Omron Sysmac Studio project 20-801-IP106 (Sysmac Studio 1.41.0.10, StandardProject)

# Controller new_Controller_0: NX1P2-1040DT version 1.41
Units and slaves: 節點1 : ASDA-A2-E CoE Drive (E001); 節點2 : ASDA-A2-E CoE Drive (E002); 節點3 : ASDA-A2-E CoE Drive (E003); 節點4 : ASDA-A2-E CoE Drive (E004)
Axis MC_AxisX, settings changed from default: AxisType=ServoType, FunctionLimit=SingleAxisPTP, UnitsConversion=EnumElement2, UnitsNumerator=1280000, UnitsDenominator=20, MaxVelocity=1500, MaxJogVelocity=150, InPositionBand=1, InPositionCheckTime=100, ZeroPositionBand=0.01, HomingMode=LimitOnly, StartDirection=NegativeDirection, HomingVelocity=10, HomingApproachVelocity=5, OriginCompensationValue=1, CompensationVelocity=5
Axis MC_AxisY, settings changed from default: AxisNumber=1, AxisType=ServoType, FunctionLimit=SingleAxisPTP, UnitsConversion=EnumElement2, UnitsNumerator=1280000, UnitsDenominator=20, MaxVelocity=1500, MaxJogVelocity=150, InPositionBand=1, InPositionCheckTime=100, ZeroPositionBand=0.01, HomingMode=LimitOnly, StartDirection=NegativeDirection, HomingVelocity=10, HomingApproachVelocity=5, OriginCompensationValue=1, CompensationVelocity=5
Axis MC_AxisZ, settings changed from default: AxisNumber=2, AxisType=ServoType, FunctionLimit=SingleAxisPTP, UnitsConversion=EnumElement2, UnitsNumerator=1280000, UnitsDenominator=20, MaxVelocity=1500, MaxJogVelocity=150, InPositionBand=1, InPositionCheckTime=100, ZeroPositionBand=0.01, HomingMode=LimitOnly, StartDirection=NegativeDirection, HomingVelocity=10, HomingApproachVelocity=5, OriginCompensationValue=1, CompensationVelocity=5
Axis MC_AxisS, settings changed from default: AxisNumber=3, AxisType=ServoType, UnitsConversion=EnumElement5, UnitsNumerator=1280000, UnitsDenominator=120, TravelDistancePerWorkRotation=360, WorkGearRatio=3, MaxVelocity=18000, MaxJogVelocity=1800, InPositionBand=0.1, InPositionCheckTime=500, ZeroPositionBand=0.05, HomingVelocity=100, HomingApproachVelocity=50
Task PrimaryTask (priority 4, period or condition 2000): prAxisDefineX, prAxisDefineY, prAxisDefineZ, prAxisDefineS, prCommProgram, prError, prInitialize, prScrewData, prBZAndLight, prBowlFeeder, prCycleTime, prMain, prScrewFlow, prFeedScrew

TYPE stScrewData : STRUCT
    PositionX : array[0..29] of lreal;
    PositionY : array[0..29] of lreal;
    PositionZ : array[0..29] of lreal;
    IsLastPoint : array[0..29] of bool;
END_STRUCT END_TYPE
TYPE AxisShow : STRUCT
    bHomed : BOOL;
END_STRUCT END_TYPE

VAR_GLOBAL CONSTANT
    MC_AxisX : _sAXIS_REF;  (* at MC://_MC_AX[0] *)
    MC_AxisY : _sAXIS_REF;  (* at MC://_MC_AX[1] *)
    MC_AxisZ : _sAXIS_REF;  (* at MC://_MC_AX[2] *)
    MC_AxisS : _sAXIS_REF;  (* at MC://_MC_AX[3] *)
END_VAR
VAR_GLOBAL
    PB_Start : BOOL;  (* at BuiltInIO://cpu/#0/Input_Bit_00; published *)
    PB_Reset : BOOL;  (* at BuiltInIO://cpu/#0/Input_Bit_01; published *)
    PB_ESTOP : BOOL;  (* at BuiltInIO://cpu/#0/Input_Bit_02; published *)
    LS_UpDownBack : BOOL;  (* at BuiltInIO://cpu/#0/Input_Bit_03; published *)
    LS_UpDownOut : BOOL;  (* at BuiltInIO://cpu/#0/Input_Bit_04; published *)
    LS_THBack : BOOL;  (* at BuiltInIO://cpu/#0/Input_Bit_05; published *)
    LS_THOut : BOOL;  (* at BuiltInIO://cpu/#0/Input_Bit_06; published *)
    SNR_AirSource : BOOL;  (* at BuiltInIO://cpu/#0/Input_Bit_07; published *)
    SNR_FeedScrew : BOOL;  (* at BuiltInIO://cpu/#0/Input_Bit_08; published *)
    SNR_BowlFeeder : BOOL;  (* at BuiltInIO://cpu/#0/Input_Bit_09; published *)
    SNR_InPositionCheck : BOOL;  (* at BuiltInIO://cpu/#0/Input_Bit_10; published *)
    SOL_UpDown : BOOL;  (* at BuiltInIO://cpu/#0/Output_Bit_00; published *)
    SOL_TH : BOOL;  (* at BuiltInIO://cpu/#0/Output_Bit_01; published *)
    SOL_Fix : BOOL;  (* at BuiltInIO://cpu/#0/Output_Bit_02; published *)
    SOL_FeedScrew : BOOL;  (* at BuiltInIO://cpu/#0/Output_Bit_03; published *)
    BZ : BOOL;  (* at BuiltInIO://cpu/#0/Output_Bit_04; published *)
    YL : BOOL;  (* at BuiltInIO://cpu/#0/Output_Bit_10; published *)
    GL : BOOL;  (* at BuiltInIO://cpu/#0/Output_Bit_06; published *)
    RL : BOOL;  (* at BuiltInIO://cpu/#0/Output_Bit_07; published *)
    RY_BowlFeeder : BOOL;  (* at BuiltInIO://cpu/#0/Output_Bit_08; published *)
    RY_BrakeAxisZ : BOOL;  (* at BuiltInIO://cpu/#0/Output_Bit_09; published *)
    RY_BowlFeederMotor : BOOL;  (* at IOBus://unit#3/Output Bit 16 bits/Output Bit 00; published *)
    AutoStatus : BOOL;  (* published *)
    HMIPB_AllSerchHome : BOOL;  (* published *)
    HMIPB_UpDown : BOOL;  (* published *)
    HMIPB_TH : BOOL;  (* published *)
    HMIPB_Fix : BOOL;  (* published *)
    HMIPB_ScrewMode_Torque : BOOL;  (* 鎖付方式(扭力/位置); published *)
    HMIPB_FeedScrew : BOOL;  (* published *)
    HMIPB_HighSpeed : BOOL;  (* published *)
    HMIPB_AlarmResetAxisX : BOOL;  (* published *)
    HMIPB_AlarmResetAxisY : BOOL;  (* published *)
    HMIPB_AlarmResetAxisZ : BOOL;  (* published *)
    HMIPB_AlarmResetAxisS : BOOL;  (* published *)
    HMIPB_ServoStopAxisX : BOOL;  (* published *)
    HMIPB_ServoStopAxisY : BOOL;  (* published *)
    HMIPB_ServoStopAxisZ : BOOL;  (* published *)
    HMIPB_ServoStopAxisS : BOOL;  (* published *)
    HMIPB_FW_AxisX : BOOL;  (* published *)
    HMIPB_RW_AxisX : BOOL;  (* published *)
    HMIPB_FW_AxisY : BOOL;  (* published *)
    HMIPB_RW_AxisY : BOOL;  (* published *)
    HMIPB_FW_AxisZ : BOOL;  (* published *)
    HMIPB_RW_AxisZ : BOOL;  (* published *)
    HMIPB_FW_AxisS : BOOL;  (* published *)
    HMIPB_RW_AxisS : BOOL;  (* published *)
    HMIPB_ServoON_AxisX : BOOL;  (* published *)
    HMIPB_ServoON_AxisY : BOOL;  (* published *)
    HMIPB_ServoON_AxisZ : BOOL;  (* published *)
    HMIPB_ServoON_AxisS : BOOL;  (* published *)
    HMIPB_SerchHome_AxisX : BOOL;  (* published *)
    HMIPB_SerchHome_AxisY : BOOL;  (* published *)
    HMIPB_SerchHome_AxisZ : BOOL;  (* published *)
    HMIPB_SerchHome_AxisS : BOOL;  (* published *)
    HMIPB_MoveAbs_AxisX : BOOL;  (* published *)
    HMIPB_MoveAbs_AxisY : BOOL;  (* published *)
    HMIPB_MoveAbs_AxisZ : BOOL;  (* published *)
    HMIPB_GoZero_AxisX : BOOL;  (* published *)
    HMIPB_GoZero_AxisY : BOOL;  (* published *)
    HMIPB_GoZero_AxisZ : BOOL;  (* published *)
    HMIPB_MoveAbs_TechX : BOOL;  (* published *)
    HMIPB_MoveAbs_TechY : BOOL;  (* published *)
    HMIPB_MoveAbs_TechZ : BOOL;  (* published *)
    HMIPB_ResetCount : BOOL;  (* published *)
    HMIPB_BrakeAxisZ : BOOL;  (* published *)
    ReadScrewData : BOOL;  (* published *)
    WriteScrewData : BOOL;  (* published *)
    SetPointData : BOOL;  (* published *)
    Error_PB_ESTOP : BOOL;  (* published *)
    Error_LS_UpDownBack : BOOL;  (* published *)
    Error_LS_UpDownOut : BOOL;  (* published *)
    Error_LS_THBack : BOOL;  (* published *)
    Error_LS_THOut : BOOL;  (* published *)
    Error_SNR_AirSource : BOOL;  (* published *)
    Error_SNR_FeedScrew : BOOL;  (* published *)
    Error_SNR_BowlFeeder : BOOL;  (* published *)
    Error_AxisX : BOOL;  (* published *)
    Error_AxisY : BOOL;  (* published *)
    Error_AxisZ : BOOL;  (* published *)
    Error_AxisS : BOOL;  (* published *)
    Flash1s : BOOL;
    SystemReadyStatus : BOOL;
    ErrorStatus_MachineStop : BOOL;  (* published *)
    ErrorStatus_MachineNonStop : BOOL;  (* published *)
    MachineRunning : BOOL;  (* published *)
    UP_InitialFlag : BOOL;
    FixOff_InitialFlag : BOOL;
    ScrewStopFlag : BOOL;
    SerchHomeAxisX_InitialFlag : BOOL;
    SerchHomeAxisY_InitialFlag : BOOL;
    SerchHomeAxisZ_InitialFlag : BOOL;
    SerchHomeAxisS_InitialFlag : BOOL;
    GoZeroAxisX_InitialFlag : BOOL;
    GoZeroAxisY_InitialFlag : BOOL;
    GoZeroAxisZ_InitialFlag : BOOL;
    Main2ScrewFlag : BOOL;  (* Main發screw開始flag *)
    Main2FeedScrewFlag : BOOL;  (* Main發送螺絲開始flag *)
    Main2DownFlag : BOOL;
    Main2UpFlag : BOOL;
    FeedScrewErrorFlag : BOOL;
    ResetFeedScrewErrorFlag : BOOL;
    ScrewNGFlag : BOOL;
END_VAR
VAR_GLOBAL RETAIN
    ScrewDatas : array[0..39] of stscrewdata;
    HMI_ItemNotExistsDelayTime : LINT;  (* published *)
    HMI_ItemExistsDelayTime : LINT;  (* published *)
    HMI_ItemNotExistsErrorTime : LINT;  (* published *)
    HMI_FeedScrewTime : LINT;  (* published *)
    HMI_CheckOKTime : LINT;  (* 滑牙計時OK; published *)
    HMI_CheckNGTime : LINT;  (* 滑牙計時NG; published *)
    HMI_AutoSpeedXY : LREAL;  (* mm/s; published *)
    HMI_AutoSpeedZ : LREAL;  (* mm/s; published *)
    HMI_HighSpeed : LREAL;  (* mm/s; published *)
    HMI_LowSpeed : LREAL;  (* mm/s; published *)
    HMI_ScrewSpeed : LREAL;  (* RPM; published *)
    HMI_ScrewTorque : LREAL;  (* %; published *)
END_VAR
VAR_GLOBAL
    HMI_Acc : LREAL;
    HMI_Dec : LREAL;
    HMI_Jerk : LREAL;
END_VAR
VAR_GLOBAL RETAIN
    HMI_JobNo : INT;  (* published *)
    HMI_PointNo : INT;  (* published *)
    HMI_AllCount : UDINT;  (* published *)
END_VAR
VAR_GLOBAL
    HMI_CycleTime : LINT;  (* published *)
END_VAR
VAR_GLOBAL RETAIN
    HMI_BackoutD : LREAL;  (* published *)
    ScrewInClip : INT;
    OilPointX : LREAL;  (* published *)
    OilPointY : LREAL;  (* published *)
    OilPointZ : LREAL;  (* published *)
END_VAR
VAR_GLOBAL
    PositionX : ARRAY[0..29] of lreal;  (* published *)
    PositionY : ARRAY[0..29] of lreal;  (* published *)
    PositionZ : ARRAY[0..29] of lreal;  (* published *)
    LastScrewPoint : ARRAY[0..29] of bool;  (* published *)
    ShowOKs : ARRAY[0..29] of bool;  (* published *)
    ShowNGs : ARRAY[0..29] of bool;  (* published *)
    Homed_ShowAixs : array[0..3] of bool;  (* published *)
    Error_ShowAixs : array[0..3] of bool;  (* published *)
    POT_ShowAxis : array[0..3] of bool;  (* published *)
    NOT_ShowAxis : array[0..3] of bool;  (* published *)
    CurrentPostion_ShowAxis : array[0..3] of lreal;  (* published *)
    CurrentSpeed_ShowAxis : array[0..3] of lreal;  (* published *)
    CurrentTorque_ShowAxis : array[0..3] of lreal;  (* published *)
    SOL_BowlFeederBlow : BOOL;  (* at IOBus://unit#3/Output Bit 16 bits/Output Bit 01 *)
END_VAR

PROGRAM prCommProgram
VAR
    statusFlash1s : BOOL;
    bClock : BOOL;
    TON1 : TON;
    TON2 : TON;
    R_TRIG1 : R_TRIG;
END_VAR
VAR_EXTERNAL
    Flash1s : BOOL;
    HMIPB_ResetCount : BOOL;
    HMI_AllCount : UDINT;
END_VAR
//bClock:=Get1sClk();
IF HMIPB_ResetCount THEN
	HMI_AllCount:=0;
END_IF;
//flsash 1s
TON1(In:=NOT(statusFlash1s), PT:=t#1s);
TON2(In:=(statusFlash1s), PT:=t#1s);
IF TON1.Q THEN
	bClock:=TRUE;
END_IF;
IF TON2.Q THEN
	bClock:=FALSE;
END_IF;
Flash1s:=bClock;
statusFlash1s:=Flash1s;
END_PROGRAM

PROGRAM prBowlFeeder
VAR
    bowlfedder1 : BowlFeeder;
END_VAR
VAR_EXTERNAL
    SNR_BowlFeeder : BOOL;
    HMI_ItemNotExistsDelayTime : LINT;
    HMI_ItemExistsDelayTime : LINT;
    HMI_ItemNotExistsErrorTime : LINT;
    RY_BowlFeeder : BOOL;
    Error_SNR_BowlFeeder : BOOL;
    SOL_BowlFeederBlow : BOOL;
    RY_BowlFeederMotor : BOOL;
END_VAR
bowlfedder1(
	bFullSNR:=SNR_BowlFeeder,
	iItemNotExistDelayTime:=HMI_ItemNotExistsDelayTime,
	iItemExistTime:=HMI_ItemExistsDelayTime,
	iItemNotExistErrorTime:=HMI_ItemNotExistsErrorTime,
	bFullSNRError=>Error_SNR_BowlFeeder);
RY_BowlFeeder:=bowlfedder1.bFullRY;
RY_BowlFeederMotor:=bowlfedder1.bFullRY;
SOL_BowlFeederBlow:=bowlfedder1.bFullRY;
END_PROGRAM

PROGRAM prInitialize
VAR
    InitFlow : INT;
    TON1 : TON;
    R_TRIG1 : R_TRIG;
    ErrorState : BOOL;
END_VAR
VAR_EXTERNAL
    ErrorStatus_MachineStop : BOOL;
    PB_Reset : BOOL;
    LS_UpDownBack : BOOL;
END_VAR
VAR_EXTERNAL CONSTANT
    MC_AxisZ : _sAXIS_REF;
    MC_AxisS : _sAXIS_REF;
    MC_AxisX : _sAXIS_REF;
    MC_AxisY : _sAXIS_REF;
END_VAR
VAR_EXTERNAL
    HMIPB_ServoON_AxisX : BOOL;
    HMIPB_ServoON_AxisY : BOOL;
    HMIPB_ServoON_AxisZ : BOOL;
    HMIPB_ServoON_AxisS : BOOL;
    SystemReadyStatus : BOOL;
    UP_InitialFlag : BOOL;
    SerchHomeAxisZ_InitialFlag : BOOL;
    GoZeroAxisZ_InitialFlag : BOOL;
    SerchHomeAxisX_InitialFlag : BOOL;
    SerchHomeAxisY_InitialFlag : BOOL;
    GoZeroAxisX_InitialFlag : BOOL;
    GoZeroAxisY_InitialFlag : BOOL;
    SerchHomeAxisS_InitialFlag : BOOL;
    FixOff_InitialFlag : BOOL;
    LS_THBack : BOOL;
    SOL_Fix : BOOL;
    HMIPB_AllSerchHome : BOOL;
    RY_BrakeAxisZ : BOOL;
    AutoStatus : BOOL;
    Error_AxisX : BOOL;
    Error_AxisY : BOOL;
    Error_AxisZ : BOOL;
    Error_AxisS : BOOL;
    Error_LS_THBack : BOOL;
    Error_LS_THOut : BOOL;
    Error_LS_UpDownBack : BOOL;
    Error_LS_UpDownOut : BOOL;
    Error_PB_ESTOP : BOOL;
    HMIPB_HighSpeed : BOOL;
    SOL_UpDown : BOOL;
    HMI_PointNo : INT;
END_VAR
//********************************************************************
//power on=0
//idle=1
//Servo On=2
//sol up=3
//up  reached=4

//Z軸未HOMED=100
//Axis Z serch home start=101
//Axis z serch home finiish=102

//Z軸已HOMED=200
//Axis Z go to 0 start=201
//Axis Z go to 0 finish=202

//X or Y軸未HOMED=300
//Axis X,Y serch home start=301
//Axis X,Y serch home finish=302

//X and Y軸已HOMED=400
//Axis X,Y go to 0 start=401
//Axis X,Y go to 0 finish=402

//Axis S serch home start=5
//Axis S serch home finish=6
//sol Fix off=7
//sol fix reached,system ready on=8
//********************************************************************
ErrorState:=
Error_AxisX OR
Error_AxisY OR
Error_AxisZ OR
Error_AxisS OR
Error_LS_THBack OR
Error_LS_THOut;
//power on=0
IF P_First_Run OR ErrorState OR R_TRIG1.Q THEN
	InitFlow:=0;
	SystemReadyStatus:=FALSE;
	AutoStatus:=FALSE;
	UP_InitialFlag:=FALSE;
	FixOff_InitialFlag:=FALSE;
	HMI_PointNo:=0;
END_IF;
//idle=1
IF InitFlow=0 AND NOT(ErrorState) THEN
	InitFlow:=1;
END_IF;
IF Error_PB_ESTOP THEN
	InitFlow:=1;
	AutoStatus:=FALSE;
	UP_InitialFlag:=FALSE;
	FixOff_InitialFlag:=FALSE;
END_IF;
//Servo On=2
R_TRIG1(Clk:=HMIPB_AllSerchHome);
TON1(In:=InitFlow=1 AND MC_AxisX.DrvStatus.MainPower AND MC_AxisY.DrvStatus.MainPower AND MC_AxisZ.DrvStatus.MainPower AND MC_AxisS.DrvStatus.MainPower, PT:=t#3s);
IF InitFlow=1 AND TON1.Q  and NOT(ErrorState) AND NOT(Error_PB_ESTOP) THEN
	HMIPB_ServoON_AxisX:=TRUE;
	HMIPB_ServoON_AxisY:=TRUE;
	HMIPB_ServoON_AxisZ:=TRUE;
	HMIPB_ServoON_AxisS:=TRUE;
	HMIPB_HighSpeed:=TRUE;
	InitFlow:=2;
END_IF;
//sol up=3
IF InitFlow=2 AND HMIPB_HighSpeed AND MC_AxisX.Status.Ready AND MC_AxisY.Status.Ready AND MC_AxisZ.Status.Ready AND MC_AxisS.Status.Ready AND RY_BrakeAxisZ THEN
	InitFlow:=3;
	UP_InitialFlag:=TRUE;
END_IF;
//up  reached=4
IF InitFlow=3 AND UP_InitialFlag AND LS_UpDownBack AND NOT(SOL_UpDown) THEN
	InitFlow:=4;
	UP_InitialFlag:=FALSE;
END_IF;
//********************************************************************
//Z軸未HOMED=100
IF InitFlow=4 AND NOT(UP_InitialFlag) AND NOT(MC_AxisZ.Details.Homed) THEN
	InitFlow:=100;
END_IF;
//Axis Z serch home start=101
IF InitFlow=100 THEN
	InitFlow:=101;
	SerchHomeAxisZ_InitialFlag:=TRUE;
END_IF;
//Axis z serch home finiish=102
IF InitFlow=101 AND NOT(SerchHomeAxisZ_InitialFlag) AND MC_AxisZ.Details.Homed THEN
	InitFlow:=102;
END_IF;
//********************************************************************
//Z軸已HOMED=200
IF InitFlow=4 AND NOT(UP_InitialFlag) AND MC_AxisZ.Details.Homed THEN
	InitFlow:=200;
END_IF;
//Axis Z go to 0 start=201
IF InitFlow=200 THEN
	InitFlow:=201;
	GoZeroAxisZ_InitialFlag:=TRUE;
END_IF;
//Axis Z go to 0 finish=202
IF InitFlow=201 AND NOT(GoZeroAxisZ_InitialFlag) AND MC_AxisZ.Details.InHome THEN
	InitFlow:=202;
END_IF;
//********************************************************************
//X or Y軸未HOMED=300
IF (InitFlow=102 OR InitFlow=202) AND (NOT(MC_AxisX.Details.Homed) OR NOT(MC_AxisY.Details.Homed)) THEN
	InitFlow:=300;
END_IF;
//Axis X,Y serch home start=301
IF InitFlow=300 THEN
	InitFlow:=301;
	SerchHomeAxisX_InitialFlag:=TRUE;
	SerchHomeAxisY_InitialFlag:=TRUE;
END_IF;
//Axis X,Y serch home finish=302
IF InitFlow=301 AND NOT(SerchHomeAxisX_InitialFlag) AND NOT(SerchHomeAxisY_InitialFlag) AND MC_AxisX.Details.Homed AND MC_AxisY.Details.Homed THEN
	InitFlow:=302;
END_IF;
//********************************************************************
//X and Y軸已HOMED=400
IF (InitFlow=102 OR InitFlow=202) AND MC_AxisX.Details.Homed AND MC_AxisY.Details.Homed THEN
	InitFlow:=400;
END_IF;
//Axis X,Y go to 0 start=401
IF InitFlow=400 THEN
	InitFlow:=401;
	GoZeroAxisX_InitialFlag:=TRUE;
	GoZeroAxisY_InitialFlag:=TRUE;
END_IF;
//Axis X,Y go to 0 finish=402
IF InitFlow=401 AND NOT(GoZeroAxisX_InitialFlag) AND NOT(GoZeroAxisY_InitialFlag) AND
	MC_AxisX.Details.InHome AND
	MC_AxisY.Details.InHome THEN
	InitFlow:=402;
END_IF;
//********************************************************************
//Axis S serch home start=5
IF InitFlow=302 AND MC_AxisX.Details.Homed  AND MC_AxisY.Details.Homed THEN
	InitFlow:=5;
	SerchHomeAxisS_InitialFlag:=TRUE;
END_IF;
IF InitFlow=402 AND MC_AxisX.Details.InHome AND MC_AxisY.Details.InHome THEN
	InitFlow:=5;
	SerchHomeAxisS_InitialFlag:=TRUE;
END_IF;
//Axis S serch home finish=6
IF InitFlow=5 AND NOT(SerchHomeAxisS_InitialFlag) AND MC_AxisS.Details.Homed THEN
	InitFlow:=6;
END_IF;
//sol Fix off=7
IF InitFlow=6 THEN
	InitFlow:=7;
	FixOff_InitialFlag:=TRUE;
END_IF;
//sol fix reached,system ready on=8
IF InitFlow=7 AND FixOff_InitialFlag AND NOT(SOL_Fix) THEN
	InitFlow:=8;
	FixOff_InitialFlag:=FALSE;
	SystemReadyStatus:=TRUE;
END_IF;
//Serch home finish=1000
IF InitFlow=8 AND SystemReadyStatus THEN
	InitFlow:=1000;
END_IF;
END_PROGRAM

PROGRAM prAxisDefineX
VAR
    MC_Power1 : MC_Power;
    MC_Reset1 : MC_Reset;
    MC_Stop1 : MC_Stop;
    MC_Home1 : MC_Home;
    MC_MoveJog1 : MC_MoveJog;
    MC_MoveAbsolute1 : MC_MoveAbsolute;
    MC_MoveAbsolute2 : MC_MoveAbsolute;
    MC_MoveAbsolute3 : MC_MoveAbsolute;
    MoveSpeed : LREAL;
    bInterlock : BOOL;
END_VAR
VAR_EXTERNAL CONSTANT
    MC_AxisX : _sAXIS_REF;
END_VAR
VAR_EXTERNAL
    HMIPB_ServoON_AxisX : BOOL;
    Error_AxisX : BOOL;
    HMIPB_SerchHome_AxisX : BOOL;
    SerchHomeAxisx_InitialFlag : BOOL;
    PB_Reset : BOOL;
    HMIPB_AlarmResetAxisX : BOOL;
    AutoStatus : BOOL;
    HMIPB_HighSpeed : BOOL;
    HMI_HighSpeed : LREAL;
    HMI_LowSpeed : LREAL;
    HMIPB_MoveAbs_AxisX : BOOL;
    GoZeroAxisX_InitialFlag : BOOL;
    HMIPB_FW_AxisX : BOOL;
    HMIPB_RW_AxisX : BOOL;
    PB_ESTOP : BOOL;
    HMIPB_ServoStopAxisX : BOOL;
    Homed_ShowAixs : array[0..3] of bool;
    Error_ShowAixs : array[0..3] of bool;
    POT_ShowAxis : array[0..3] of bool;
    NOT_ShowAxis : array[0..3] of bool;
    CurrentPostion_ShowAxis : array[0..3] of lreal;
    CurrentSpeed_ShowAxis : array[0..3] of lreal;
    CurrentTorque_ShowAxis : array[0..3] of lreal;
END_VAR
VAR_EXTERNAL CONSTANT
    MC_AxisZ : _sAXIS_REF;
END_VAR
VAR_EXTERNAL
    HMI_AutoSpeedXY : LREAL;
    HMIPB_GoZero_AxisX : BOOL;
    ScrewDatas : array[0..39] of stscrewdata;
    HMI_JobNo : INT;
    HMI_PointNo : INT;
    LS_UpDownBack : BOOL;
    SOL_UpDown : BOOL;
END_VAR
VAR_EXTERNAL CONSTANT
    _MC_ErrSta : WORD;
END_VAR
VAR_EXTERNAL
    HMI_Acc : LREAL;
    HMI_Dec : LREAL;
    HMI_Jerk : LREAL;
    HMIPB_MoveAbs_TechX : BOOL;
    PositionX : ARRAY[0..29] of lreal;
END_VAR
Error_AxisX:=MC_AxisX.DrvStatus.DrvAlarm OR MC_AxisX.DrvStatus.DrvWarning OR NOT(MC_AxisX.DrvStatus.MainPower) OR _MC_ErrSta<>0;		//Error
bInterlock:=MC_AxisX.DrvStatus.ServoOn AND MC_AxisZ.Details.Homed AND MC_AxisZ.Act.Pos>-1 AND MC_AxisZ.Act.Pos<1 AND LS_UpDownBack AND NOT(SOL_UpDown);
MC_Power1(Axis:=MC_AxisX, Enable:=HMIPB_ServoON_AxisX);		//servo on
MC_Reset1(Axis:=MC_AxisX, Execute:=HMIPB_AlarmResetAxisX OR PB_Reset);		//Alarm Reset
MC_Stop1(Axis:=MC_AxisX, Execute:=NOT(PB_ESTOP) OR HMIPB_ServoStopAxisX, Deceleration:=0, Jerk:=0, BufferMode:=_mcAborting);		//Servo Stop
MC_Home1(Axis:=MC_AxisX, Execute:=HMIPB_SerchHome_AxisX OR SerchHomeAxisx_InitialFlag);		//Serch home
MC_MoveJog1(Axis:=MC_AxisX, PositiveEnable:=HMIPB_FW_AxisX AND bInterlock, NegativeEnable:=HMIPB_RW_AxisX AND bInterlock, Velocity:=MoveSpeed, Acceleration:=0, Deceleration:=0);		//JOG
IF MC_Home1.Done OR MC_Home1.CommandAborted OR MC_Home1.Error THEN
	SerchHomeAxisX_InitialFlag:=FALSE;
END_IF;
IF AutoStatus THEN
	MoveSpeed:=HMI_AutoSpeedXY;
ELSE
	IF HMIPB_HighSpeed THEN
		MoveSpeed:=HMI_HighSpeed;
	ELSE
		MoveSpeed:=HMI_LowSpeed;
	END_IF;
END_IF;
MC_MoveAbsolute1(Axis:=MC_AxisX, Execute:=(HMIPB_GoZero_AxisX OR GoZeroAxisX_InitialFlag) AND bInterlock AND MC_AxisX.Details.Homed, Position:=0, Velocity:=MoveSpeed, Acceleration:=HMI_Acc,Deceleration:=HMI_Dec,jerk:=HMI_Jerk);		//Go Zero
IF MC_MoveAbsolute1.Done OR MC_MoveAbsolute1.Error OR MC_MoveAbsolute1.CommandAborted THEN
	GoZeroAxisX_InitialFlag:=FALSE;
END_IF;
MC_MoveAbsolute2(Axis:=MC_AxisX, Execute:=(HMIPB_MoveAbs_AxisX) AND bInterlock AND MC_AxisX.Details.Homed, Position:=ScrewDatas[HMI_JobNo].PositionX[HMI_PointNo], Velocity:=MoveSpeed, Acceleration:=HMI_Acc,Deceleration:=HMI_Dec,jerk:=HMI_Jerk);		//Go ABS
MC_MoveAbsolute3(Axis:=MC_AxisX, Execute:=(HMIPB_MoveAbs_TechX) AND bInterlock AND MC_AxisX.Details.Homed, Position:=PositionX[HMI_PointNo], Velocity:=MoveSpeed, Acceleration:=HMI_Acc,Deceleration:=HMI_Dec,jerk:=HMI_Jerk);		//Go ABS
//*****************************************************HMI Show**********************************************************************************************************
Homed_ShowAixs[0]:=MC_AxisX.Details.Homed;
Error_ShowAixs[0]:=MC_AxisX.DrvStatus.DrvAlarm OR MC_AxisX.DrvStatus.DrvWarning;
POT_ShowAxis[0]:=NOT(MC_AxisX.DrvStatus.P_OT);
NOT_ShowAxis[0]:=NOT(MC_AxisX.DrvStatus.N_OT);
CurrentPostion_ShowAxis[0]:=MC_AxisX.Act.Pos;
CurrentSpeed_ShowAxis[0]:=MC_AxisX.Act.Vel;
CurrentTorque_ShowAxis[0]:=MC_AxisX.Act.Trq;
END_PROGRAM

PROGRAM prBZAndLight
VAR_EXTERNAL CONSTANT
    MC_AxisX : _sAXIS_REF;
END_VAR
VAR_EXTERNAL
    Flash1s : BOOL;
    GL : BOOL;
    YL : BOOL;
    SystemReadyStatus : BOOL;
    ErrorStatus_MachineNonStop : BOOL;
    ErrorStatus_MachineStop : BOOL;
    RL : BOOL;
    BZ : BOOL;
    MachineRunning : BOOL;
    Error_SNR_FeedScrew : BOOL;
    ScrewNGFlag : BOOL;
END_VAR
(*BZ*)	
IF (ErrorStatus_MachineStop OR ErrorStatus_MachineNonStop OR Error_SNR_FeedScrew OR ScrewNGFlag) THEN
	BZ:=Flash1s;
	ELSE
	BZ:=FALSE;
END_IF;
//(*紅燈長亮:異常*)
IF SystemReadyStatus AND (ErrorStatus_MachineStop OR Error_SNR_FeedScrew) THEN
	RL:=TRUE;
	ELSE
	RL:=FALSE;
END_IF;
(*綠燈閃爍:運轉,長亮:待機*)
IF SystemReadyStatus AND NOT(ErrorStatus_MachineNonStop) AND NOT(ErrorStatus_MachineStop) AND NOT(Error_SNR_FeedScrew)  THEN
	IF MachineRunning THEN
		GL:=Flash1s;
	ELSE
		GL:=TRUE;
	END_IF;
	ELSE
	GL:=FALSE;
END_IF;
(*黃燈閃爍:振動筒缺料*)
IF SystemReadyStatus AND ErrorStatus_MachineNonStop AND NOT(ErrorStatus_MachineStop) THEN
	YL:=Flash1s;
	ELSE
	YL:=FALSE;
END_IF;
END_PROGRAM

PROGRAM prAxisDefineY
VAR
    MC_Power1 : MC_Power;
    MC_Reset1 : MC_Reset;
    MC_Stop1 : MC_Stop;
    MC_Home1 : MC_Home;
    MC_MoveJog1 : MC_MoveJog;
    MC_MoveAbsolute1 : MC_MoveAbsolute;
    MC_MoveAbsolute2 : MC_MoveAbsolute;
    MC_MoveAbsolute3 : MC_MoveAbsolute;
    MoveSpeed : LREAL;
    bInterlock : BOOL;
END_VAR
VAR_EXTERNAL CONSTANT
    MC_AxisY : _sAXIS_REF;
END_VAR
VAR_EXTERNAL
    HMIPB_ServoON_AxisY : BOOL;
    Error_AxisY : BOOL;
    HMIPB_SerchHome_AxisY : BOOL;
    SerchHomeAxisY_InitialFlag : BOOL;
    HMIPB_AlarmResetAxisY : BOOL;
    AutoStatus : BOOL;
    HMIPB_HighSpeed : BOOL;
    HMI_HighSpeed : LREAL;
    HMI_LowSpeed : LREAL;
    HMIPB_MoveAbs_AxisY : BOOL;
    GoZeroAxisY_InitialFlag : BOOL;
    HMIPB_FW_AxisY : BOOL;
    HMIPB_RW_AxisY : BOOL;
    PB_ESTOP : BOOL;
    HMIPB_ServoStopAxisY : BOOL;
    Homed_ShowAixs : array[0..3] of bool;
    Error_ShowAixs : array[0..3] of bool;
    POT_ShowAxis : array[0..3] of bool;
    NOT_ShowAxis : array[0..3] of bool;
    CurrentPostion_ShowAxis : array[0..3] of lreal;
    CurrentSpeed_ShowAxis : array[0..3] of lreal;
    CurrentTorque_ShowAxis : array[0..3] of lreal;
    HMIPB_ServoStopAxisX : BOOL;
END_VAR
VAR_EXTERNAL CONSTANT
    MC_AxisZ : _sAXIS_REF;
END_VAR
VAR_EXTERNAL
    HMI_AutoSpeedXY : LREAL;
    HMIPB_GoZero_AxisY : BOOL;
    ScrewDatas : array[0..39] of stscrewdata;
    HMI_JobNo : INT;
    HMI_PointNo : INT;
    LS_UpDownBack : BOOL;
    SOL_UpDown : BOOL;
    PB_Reset : BOOL;
END_VAR
VAR_EXTERNAL CONSTANT
    _MC_ErrSta : WORD;
END_VAR
VAR_EXTERNAL
    HMI_Acc : LREAL;
    HMI_Dec : LREAL;
    HMI_Jerk : LREAL;
    HMIPB_MoveAbs_TechY : BOOL;
    PositionY : ARRAY[0..29] of lreal;
END_VAR
Error_AxisY:=MC_AxisY.DrvStatus.DrvAlarm OR MC_AxisY.DrvStatus.DrvWarning OR NOT(MC_AxisY.DrvStatus.MainPower) OR _MC_ErrSta<>0;		//Error
bInterlock:=MC_AxisY.DrvStatus.ServoOn AND MC_AxisZ.Details.Homed AND MC_AxisZ.Act.Pos>-1 AND MC_AxisZ.Act.Pos<1 AND LS_UpDownBack AND NOT(SOL_UpDown);
MC_Power1(Axis:=MC_AxisY, Enable:=HMIPB_ServoON_AxisY);		//servo on
MC_Reset1(Axis:=MC_AxisY, Execute:=HMIPB_AlarmResetAxisY OR PB_Reset);		//Alarm Reset
MC_Stop1(Axis:=MC_AxisY, Execute:=NOT(PB_ESTOP) OR HMIPB_ServoStopAxisX, Deceleration:=0, Jerk:=0, BufferMode:=_mcAborting);		//Servo Stop
MC_Home1(Axis:=MC_AxisY, Execute:=HMIPB_SerchHome_AxisY OR SerchHomeAxisY_InitialFlag);		//Serch home
MC_MoveJog1(Axis:=MC_AxisY, PositiveEnable:=HMIPB_FW_AxisY AND bInterlock, NegativeEnable:=HMIPB_RW_AxisY AND bInterlock, Velocity:=MoveSpeed, Acceleration:=0, Deceleration:=0);		//JOG
IF MC_Home1.Done OR MC_Home1.CommandAborted OR MC_Home1.Error THEN
	SerchHomeAxisY_InitialFlag:=FALSE;
END_IF;
IF AutoStatus THEN
	MoveSpeed:=HMI_AutoSpeedXY;
ELSE
	IF HMIPB_HighSpeed THEN
		MoveSpeed:=HMI_HighSpeed;
	ELSE
		MoveSpeed:=HMI_LowSpeed;
	END_IF;
END_IF;
MC_MoveAbsolute1(Axis:=MC_AxisY, Execute:=(HMIPB_GoZero_AxisY OR GoZeroAxisY_InitialFlag) AND bInterlock AND MC_AxisY.Details.Homed, Position:=0, Velocity:=MoveSpeed, Acceleration:=HMI_Acc,Deceleration:=HMI_Dec,jerk:=HMI_Jerk);		//Go Zero
IF MC_MoveAbsolute1.Done OR MC_MoveAbsolute1.Error OR MC_MoveAbsolute1.CommandAborted THEN
	GoZeroAxisY_InitialFlag:=FALSE;
END_IF;
MC_MoveAbsolute2(Axis:=MC_AxisY, Execute:=(HMIPB_MoveAbs_AxisY) AND bInterlock AND MC_AxisY.Details.Homed, Position:=ScrewDatas[HMI_JobNo].PositionY[HMI_PointNo], Velocity:=MoveSpeed, Acceleration:=HMI_Acc,Deceleration:=HMI_Dec,jerk:=HMI_Jerk);		//Go ABS
MC_MoveAbsolute3(Axis:=MC_AxisY, Execute:=(HMIPB_MoveAbs_TechY) AND bInterlock AND MC_AxisY.Details.Homed, Position:=PositionY[HMI_PointNo], Velocity:=MoveSpeed, Acceleration:=HMI_Acc,Deceleration:=HMI_Dec,jerk:=HMI_Jerk);		//Go ABS
//*****************************************************HMI Show**********************************************************************************************************
Homed_ShowAixs[1]:=MC_AxisY.Details.Homed;
Error_ShowAixs[1]:=MC_AxisY.DrvStatus.DrvAlarm OR MC_AxisY.DrvStatus.DrvWarning;
POT_ShowAxis[1]:=NOT(MC_AxisY.DrvStatus.P_OT);
NOT_ShowAxis[1]:=NOT(MC_AxisY.DrvStatus.N_OT);
CurrentPostion_ShowAxis[1]:=MC_AxisY.Act.Pos;
CurrentSpeed_ShowAxis[1]:=MC_AxisY.Act.Vel;
CurrentTorque_ShowAxis[1]:=MC_AxisY.Act.Trq;
END_PROGRAM

PROGRAM prAxisDefineZ
VAR
    MC_Power1 : MC_Power;
    MC_Reset1 : MC_Reset;
    MC_Stop1 : MC_Stop;
    MC_Home1 : MC_Home;
    MC_MoveJog1 : MC_MoveJog;
    MC_MoveAbsolute1 : MC_MoveAbsolute;
    MC_MoveAbsolute2 : MC_MoveAbsolute;
    MC_MoveAbsolute3 : MC_MoveAbsolute;
    MoveSpeed : LREAL;
    bInterlock : BOOL;
    R_TRIG1 : R_TRIG;
    F_TRIG1 : F_TRIG;
    SingleSolRy1 : SingleSolRy;
END_VAR
VAR_EXTERNAL CONSTANT
    MC_AxisZ : _sAXIS_REF;
END_VAR
VAR_EXTERNAL
    HMIPB_ServoON_AxisZ : BOOL;
    Error_AxisZ : BOOL;
    MachineRunning : BOOL;
    HMIPB_SerchHome_AxisZ : BOOL;
    SerchHomeAxisZ_InitialFlag : BOOL;
    HMIPB_MoveAbs_AxisZ : BOOL;
    AutoStatus : BOOL;
    HMIPB_HighSpeed : BOOL;
    HMI_HighSpeed : LREAL;
    HMI_LowSpeed : LREAL;
    GoZeroAxisZ_InitialFlag : BOOL;
    HMIPB_AlarmResetAxisZ : BOOL;
    HMIPB_FW_AxisZ : BOOL;
    HMIPB_RW_AxisZ : BOOL;
    PB_ESTOP : BOOL;
    HMIPB_ServoStopAxisZ : BOOL;
    RY_BrakeAxisZ : BOOL;
    Homed_ShowAixs : array[0..3] of bool;
    Error_ShowAixs : array[0..3] of bool;
    POT_ShowAxis : array[0..3] of bool;
    NOT_ShowAxis : array[0..3] of bool;
    CurrentPostion_ShowAxis : array[0..3] of lreal;
    CurrentSpeed_ShowAxis : array[0..3] of lreal;
    CurrentTorque_ShowAxis : array[0..3] of lreal;
    HMIPB_ServoStopAxisX : BOOL;
END_VAR
VAR_EXTERNAL CONSTANT
    MC_AxisX : _sAXIS_REF;
    MC_AxisY : _sAXIS_REF;
END_VAR
VAR_EXTERNAL
    HMI_AutoSpeedZ : LREAL;
    HMIPB_GoZero_AxisZ : BOOL;
    ScrewDatas : array[0..39] of stscrewdata;
    HMI_JobNo : INT;
    HMI_PointNo : INT;
    PB_Reset : BOOL;
END_VAR
VAR_EXTERNAL CONSTANT
    _MC_ErrSta : WORD;
END_VAR
VAR_EXTERNAL
    HMIPB_BrakeAxisZ : BOOL;
    HMIPB_MoveAbs_TechZ : BOOL;
    PositionZ : ARRAY[0..29] of lreal;
END_VAR
R_TRIG1(Clk:=MC_AxisZ.DrvStatus.ServoOn);
F_TRIG1(Clk:=MC_AxisZ.DrvStatus.ServoOn);
SingleSolRy1(
	inPushButton:=HMIPB_BrakeAxisZ,
	inAutoStatus:=AutoStatus,
	inAutoFlowSet:=R_TRIG1.Q,
	inAutoFlowReset:=F_TRIG1.Q,
	inInterLockBack:=TRUE,
	inInterLockOut:=TRUE,
	outSol=>RY_BrakeAxisZ);

Error_AxisZ:=MC_AxisZ.DrvStatus.DrvAlarm OR MC_AxisZ.DrvStatus.DrvWarning OR NOT(MC_AxisZ.DrvStatus.MainPower) OR _MC_ErrSta<>0;		//Error
bInterlock:=MC_AxisZ.DrvStatus.ServoOn AND RY_BrakeAxisZ AND MC_AxisX.Status.Standstill AND MC_AxisY.Status.Standstill;
MC_Power1(Axis:=MC_AxisZ, Enable:=HMIPB_ServoON_AxisZ);		//servo on
MC_Reset1(Axis:=MC_AxisZ, Execute:=HMIPB_AlarmResetAxisZ OR PB_Reset);		//Alarm Reset
MC_Stop1(Axis:=MC_AxisZ, Execute:=NOT(PB_ESTOP) OR HMIPB_ServoStopAxisX, Deceleration:=0, Jerk:=0, BufferMode:=_mcAborting);		//Servo Stop
MC_Home1(Axis:=MC_AxisZ, Execute:=HMIPB_SerchHome_AxisZ OR SerchHomeAxisZ_InitialFlag);		//Serch home
MC_MoveJog1(Axis:=MC_AxisZ, PositiveEnable:=HMIPB_FW_AxisZ AND bInterlock, NegativeEnable:=HMIPB_RW_AxisZ AND bInterlock, Velocity:=MoveSpeed, Acceleration:=0, Deceleration:=0);		//JOG
IF MC_Home1.Done OR MC_Home1.CommandAborted OR MC_Home1.Error THEN
	SerchHomeAxisZ_InitialFlag:=FALSE;
END_IF;
IF AutoStatus THEN
	MoveSpeed:=HMI_AutoSpeedZ;
ELSE
	IF HMIPB_HighSpeed THEN
		MoveSpeed:=HMI_HighSpeed;
	ELSE
		MoveSpeed:=HMI_LowSpeed;
	END_IF;
END_IF;
MC_MoveAbsolute1(Axis:=MC_AxisZ, Execute:=(HMIPB_GoZero_AxisZ OR GoZeroAxisZ_InitialFlag) AND bInterlock AND MC_AxisZ.Details.Homed, Position:=0, Velocity:=MoveSpeed);		//Go Zero
IF MC_MoveAbsolute1.Done OR MC_MoveAbsolute1.Error OR MC_MoveAbsolute1.CommandAborted THEN
	GoZeroAxisZ_InitialFlag:=FALSE;
END_IF;
MC_MoveAbsolute2(Axis:=MC_AxisZ, Execute:=(HMIPB_MoveAbs_AxisZ) AND bInterlock AND MC_AxisZ.Details.Homed, Position:=ScrewDatas[HMI_JobNo].PositionZ[HMI_PointNo], Velocity:=MoveSpeed);		//Go ABS
MC_MoveAbsolute3(Axis:=MC_AxisZ, Execute:=(HMIPB_MoveAbs_TechZ) AND bInterlock AND MC_AxisY.Details.Homed, Position:=PositionZ[HMI_PointNo], Velocity:=MoveSpeed);		//Go ABS
//*****************************************************HMI Show**********************************************************************************************************
Homed_ShowAixs[2]:=MC_AxisZ.Details.Homed;
Error_ShowAixs[2]:=MC_AxisZ.DrvStatus.DrvAlarm OR MC_AxisZ.DrvStatus.DrvWarning;
POT_ShowAxis[2]:=NOT(MC_AxisZ.DrvStatus.P_OT);
NOT_ShowAxis[2]:=NOT(MC_AxisZ.DrvStatus.N_OT);
CurrentPostion_ShowAxis[2]:=MC_AxisZ.Act.Pos;
CurrentSpeed_ShowAxis[2]:=MC_AxisZ.Act.Vel;
CurrentTorque_ShowAxis[2]:=MC_AxisZ.Act.Trq;
END_PROGRAM

PROGRAM prAxisDefineS
VAR
    MC_Power1 : MC_Power;
    MC_Reset1 : MC_Reset;
    MC_Stop1 : MC_Stop;
    MC_Home1 : MC_Home;
    MC_TorqueControl1 : MC_TorqueControl;
    MC_TorqueControl2 : MC_TorqueControl;
    TorqueValue : LREAL;
    SpeedValue : LREAL;
    F_TRIG1 : F_TRIG;
    F_TRIG2 : F_TRIG;
END_VAR
VAR_EXTERNAL CONSTANT
    MC_AxisS : _sAXIS_REF;
END_VAR
VAR_EXTERNAL
    HMIPB_ServoON_AxisS : BOOL;
    Error_AxisS : BOOL;
    HMIPB_SerchHome_AxisS : BOOL;
    SerchHomeAxisS_InitialFlag : BOOL;
    HMIPB_AlarmResetAxisS : BOOL;
    HMIPB_FW_AxisS : BOOL;
    HMIPB_RW_AxisS : BOOL;
    HMI_ScrewSpeed : LREAL;
    PB_ESTOP : BOOL;
    HMIPB_ServoStopAxisS : BOOL;
    HMI_ScrewTorque : LREAL;
    ScrewStopFlag : BOOL;
    Homed_ShowAixs : array[0..3] of bool;
    Error_ShowAixs : array[0..3] of bool;
    POT_ShowAxis : array[0..3] of bool;
    NOT_ShowAxis : array[0..3] of bool;
    CurrentPostion_ShowAxis : array[0..3] of lreal;
    CurrentSpeed_ShowAxis : array[0..3] of lreal;
    CurrentTorque_ShowAxis : array[0..3] of lreal;
    HMIPB_ServoStopAxisX : BOOL;
    PB_Reset : BOOL;
END_VAR
VAR_EXTERNAL CONSTANT
    _MC_ErrSta : WORD;
END_VAR
Error_AxisS:=MC_AxisS.DrvStatus.DrvAlarm OR MC_AxisS.DrvStatus.DrvWarning OR NOT(MC_AxisS.DrvStatus.MainPower) OR _MC_ErrSta<>0;		//Error
MC_Power1(Axis:=MC_AxisS, Enable:=HMIPB_ServoON_AxisS);		//servo on
MC_Reset1(Axis:=MC_AxisS, Execute:=HMIPB_AlarmResetAxisS OR PB_Reset);		//Alarm Reset
MC_Stop1(Axis:=MC_AxisS, Execute:=NOT(PB_ESTOP) OR HMIPB_ServoStopAxisX OR F_TRIG1.Q OR F_TRIG2.Q OR ScrewStopFlag, Deceleration:=0, Jerk:=0, BufferMode:=_mcAborting);		//Servo Stop
MC_Home1(Axis:=MC_AxisS, Execute:=HMIPB_SerchHome_AxisS OR SerchHomeAxisS_InitialFlag);		//Serch home
IF MC_Home1.Done OR MC_Home1.CommandAborted OR MC_Home1.Error THEN
	SerchHomeAxisS_InitialFlag:=FALSE;
END_IF;
TorqueValue:=HMI_ScrewTorque;
SpeedValue:=HMI_ScrewSpeed/360;
F_TRIG1(Clk:=HMIPB_FW_AxisS);
F_TRIG2(Clk:=HMIPB_RW_AxisS);
MC_TorqueControl1(Axis:=MC_AxisS, Execute:=HMIPB_FW_AxisS, Torque:=TorqueValue, TorqueRamp:=0, Velocity:=SpeedValue, Direction:=_mcPositiveDirection, BufferMode:=_mcAborting);		//JOG
MC_TorqueControl2(Axis:=MC_AxisS, Execute:=HMIPB_RW_AxisS, Torque:=TorqueValue, TorqueRamp:=0, Velocity:=SpeedValue, Direction:=_mcNegativeDirection, BufferMode:=_mcAborting);		//JOG
//*****************************************************HMI Show**********************************************************************************************************
Homed_ShowAixs[3]:=MC_AxisS.Details.Homed;
Error_ShowAixs[3]:=MC_AxisS.DrvStatus.DrvAlarm OR MC_AxisS.DrvStatus.DrvWarning;
POT_ShowAxis[3]:=NOT(MC_AxisS.DrvStatus.P_OT);
NOT_ShowAxis[3]:=NOT(MC_AxisS.DrvStatus.N_OT);
CurrentPostion_ShowAxis[3]:=MC_AxisS.Act.Pos;
CurrentSpeed_ShowAxis[3]:=MC_AxisS.Act.Vel;
CurrentTorque_ShowAxis[3]:=MC_AxisS.Act.Trq;
END_PROGRAM

PROGRAM prError
VAR
    ErrorSol1 : fbErrorSOL_S;
    ErrorSol2 : fbErrorSOL_S;
END_VAR
VAR_EXTERNAL
    ErrorStatus_MachineStop : BOOL;
    Error_AxisX : BOOL;
    Error_AxisY : BOOL;
    Error_AxisZ : BOOL;
    Error_AxisS : BOOL;
    Error_LS_THBack : BOOL;
    Error_LS_THOut : BOOL;
    Error_LS_UpDownBack : BOOL;
    Error_LS_UpDownOut : BOOL;
    Error_PB_ESTOP : BOOL;
    Error_SNR_AirSource : BOOL;
    Error_SNR_FeedScrew : BOOL;
    ErrorStatus_MachineNonStop : BOOL;
    Error_SNR_BowlFeeder : BOOL;
END_VAR
VAR_EXTERNAL CONSTANT
    _MC_ErrSta : WORD;
END_VAR
VAR_EXTERNAL
    PB_ESTOP : BOOL;
    PB_Reset : BOOL;
    AutoStatus : BOOL;
    SOL_UpDown : BOOL;
    LS_UpDownBack : BOOL;
    LS_UpDownOut : BOOL;
    SOL_TH : BOOL;
    LS_THBack : BOOL;
    LS_THOut : BOOL;
END_VAR
ErrorSol1(
	bAutoStatus:=AutoStatus,
	bResetPB:=PB_Reset,
	bSOL:=SOL_UpDown,
	bBackLS:=LS_UpDownBack,
	bOutLS:=LS_UpDownOut,
	bErrorStatus_Back=>Error_LS_UpDownBack,
	bErrorStatus_Out=>Error_LS_UpDownOut);
(*ErrorSol2(
	bAutoStatus:=AutoStatus,
	bResetPB:=PB_Reset,
	bSOL:=SOL_TH,
	bBackLS:=LS_THBack,
	bOutLS:=LS_THOut,
	bErrorStatus_Back=>Error_LS_THBack,
	bErrorStatus_Out=>Error_LS_THOut);*)
//***************************************************************
//機器停止異常
//***************************************************************
ErrorStatus_MachineStop:=
Error_AxisX OR
Error_AxisY OR
Error_AxisZ OR
Error_AxisS OR
Error_LS_THBack OR
Error_LS_THOut OR
Error_LS_UpDownBack OR
Error_LS_UpDownOut OR
Error_PB_ESTOP;
//***************************************************************
//機器不停止異常
//***************************************************************
ErrorStatus_MachineNonStop:=
Error_SNR_AirSource OR
Error_SNR_BowlFeeder;
//***************************************************************
IF NOT(PB_ESTOP) THEN
	Error_PB_ESTOP:=TRUE;
END_IF;
IF PB_Reset THEN
	Error_PB_ESTOP:=FALSE;
END_IF;
END_PROGRAM

PROGRAM prScrewData
VAR
    i : INT;
END_VAR
VAR_EXTERNAL
    ReadScrewData : BOOL;
    ScrewDatas : array[0..39] of stscrewdata;
    HMI_JobNo : INT;
    PositionX : ARRAY[0..29] of lreal;
    PositionY : ARRAY[0..29] of lreal;
    PositionZ : ARRAY[0..29] of lreal;
    WriteScrewData : BOOL;
    LastScrewPoint : ARRAY[0..29] of bool;
    SetPointData : BOOL;
END_VAR
VAR_EXTERNAL CONSTANT
    MC_AxisX : _sAXIS_REF;
END_VAR
VAR_EXTERNAL
    HMI_PointNo : INT;
END_VAR
VAR_EXTERNAL CONSTANT
    MC_AxisY : _sAXIS_REF;
    MC_AxisZ : _sAXIS_REF;
END_VAR
IF ReadScrewData THEN
	FOR i:=0 TO 29 BY 1 DO
	    PositionX[i]:=ScrewDatas[HMI_JobNo].PositionX[i];
		PositionY[i]:=ScrewDatas[HMI_JobNo].PositionY[i];
		PositionZ[i]:=ScrewDatas[HMI_JobNo].PositionZ[i];
		LastScrewPoint[i]:=ScrewDatas[HMI_JobNo].IsLastPoint[i];
	END_FOR;
	ReadScrewData:=FALSE;
END_IF;

IF WriteScrewData THEN
	FOR i:=0 TO 29 BY 1 DO
	    ScrewDatas[HMI_JobNo].PositionX[i]:=PositionX[i];
		ScrewDatas[HMI_JobNo].PositionY[i]:=PositionY[i];
		ScrewDatas[HMI_JobNo].PositionZ[i]:=PositionZ[i];
		ScrewDatas[HMI_JobNo].IsLastPoint[i]:=LastScrewPoint[i];
	END_FOR;
	WriteScrewData:=FALSE;
END_IF;

//set point
IF SetPointData THEN
	PositionX[HMI_PointNo]:= MC_AxisX.Act.Pos;
	PositionY[HMI_PointNo]:= MC_AxisY.Act.Pos;
	PositionZ[HMI_PointNo]:= MC_AxisZ.Act.Pos;
END_IF;
END_PROGRAM

PROGRAM prCycleTime
VAR
    TON1 : TON;
    tCycleTime : TIME;
END_VAR
VAR_EXTERNAL
    MachineRunning : BOOL;
    HMI_CycleTime : LINT;
END_VAR
TON1(In:=MachineRunning, PT:=t#1m,ET=>tCycleTime);
IF MachineRunning THEN
	HMI_CycleTime:=TimeToNanoSec(tCycleTime)/10000000;
END_IF;
END_PROGRAM

PROGRAM prMain
VAR
    AutoFlow : INT;
    fbSol1 : SingleSolRy;
    ErrorState : BOOL;
    MC_MoveAbsolute1 : MC_MoveAbsolute;
    MC_MoveAbsolute2 : MC_MoveAbsolute;
    MC_MoveAbsolute3 : MC_MoveAbsolute;
    MC_MoveAbsolute4 : MC_MoveAbsolute;
    MC_MoveAbsolute5 : MC_MoveAbsolute;
    MC_MoveAbsolute6 : MC_MoveAbsolute;
    MC_MoveAbsolute7 : MC_MoveAbsolute;
    MC_MoveAbsolute8 : MC_MoveAbsolute;
    MC_MoveAbsolute9 : MC_MoveAbsolute;
    bInterlockXY : BOOL;
    bInterlockZ : BOOL;
    iv : INT;
    TON1 : TON;
    TON2 : TON;
    TON3 : TON;
    TON4 : TON;
    accdec : LREAL;
    accdecY : LREAL;
    jerk : LREAL;
    feedcount : INT;
    jValue : INT;
    R_TRIG1 : R_TRIG;
    RunStatus : BOOL;
END_VAR
VAR_EXTERNAL
    HMIPB_Fix : BOOL;
    AutoStatus : BOOL;
    SOL_Fix : BOOL;
    FixOff_InitialFlag : BOOL;
    SystemReadyStatus : BOOL;
    Error_AxisX : BOOL;
    Error_AxisY : BOOL;
    Error_AxisZ : BOOL;
    Error_AxisS : BOOL;
    Error_SNR_FeedScrew : BOOL;
    Error_PB_ESTOP : BOOL;
    Main2FeedScrewFlag : BOOL;
    Main2ScrewFlag : BOOL;
    LS_UpDownBack : BOOL;
    SOL_UpDown : BOOL;
END_VAR
VAR_EXTERNAL CONSTANT
    MC_AxisZ : _sAXIS_REF;
    MC_AxisX : _sAXIS_REF;
END_VAR
VAR_EXTERNAL
    ScrewDatas : array[0..39] of stscrewdata;
    HMI_JobNo : INT;
    HMI_PointNo : INT;
    HMI_AutoSpeedXY : LREAL;
    OilPointX : LREAL;
END_VAR
VAR_EXTERNAL CONSTANT
    MC_AxisY : _sAXIS_REF;
END_VAR
VAR_EXTERNAL
    OilPointY : LREAL;
    OilPointZ : LREAL;
    HMI_AutoSpeedZ : LREAL;
    PB_Start : BOOL;
    ShowOKs : ARRAY[0..29] of bool;
    ShowNGs : ARRAY[0..29] of bool;
    LS_UpDownOut : BOOL;
    Error_LS_UpDownBack : BOOL;
    Error_LS_UpDownOut : BOOL;
    Error_SNR_AirSource : BOOL;
    Error_LS_THBack : BOOL;
    Error_LS_THOut : BOOL;
    MachineRunning : BOOL;
    Main2DownFlag : BOOL;
    Main2UpFlag : BOOL;
    HMI_AllCount : UDINT;
    HMI_FeedScrewTime : LINT;
    RY_BrakeAxisZ : BOOL;
    HMI_Acc : LREAL;
    HMI_Dec : LREAL;
    HMI_Jerk : LREAL;
    FeedScrewErrorFlag : BOOL;
    ResetFeedScrewErrorFlag : BOOL;
    PB_Reset : BOOL;
    ScrewNGFlag : BOOL;
END_VAR
//********************************************************************
//Manual
//********************************************************************
//fix sol
fbSol1(
	HMIPB_Fix,
	AutoStatus,
	AutoFlow=2,
	AutoFlow=202 OR FixOff_InitialFlag OR AutoFlow=405,
	TRUE,
	TRUE,
	SOL_Fix);
//*******************************************************************
//Auto
//********************************************************************
bInterlockXY:=
MC_AxisX.Details.Homed AND
MC_AxisX.DrvStatus.ServoOn AND
MC_AxisY.Details.Homed AND
MC_AxisY.DrvStatus.ServoOn AND
MC_AxisZ.Details.Homed AND
MC_AxisZ.Act.Pos>-1 AND
MC_AxisZ.Act.Pos<1 AND
LS_UpDownBack AND
NOT(SOL_UpDown);
bInterlockZ:=
RY_BrakeAxisZ AND
MC_AxisZ.Details.Homed AND
MC_AxisZ.DrvStatus.ServoOn AND
MC_AxisX.Status.Standstill AND
MC_AxisY.Status.Standstill;

HMI_Acc:=HMI_AutoSpeedXY/0.1;
HMI_Dec:=HMI_AutoSpeedXY/0.1;
HMI_Jerk:=HMI_Acc/0.8;
MC_MoveAbsolute1(Axis:=MC_AxisX, Execute:=(AutoFlow=10 OR AutoFlow=201) AND bInterlockXY, Position:=OilPointX, Velocity:=HMI_AutoSpeedXY, Acceleration:=HMI_Acc,Deceleration:=HMI_Dec,jerk:=HMI_Jerk);		//Go Oil
MC_MoveAbsolute2(Axis:=MC_AxisY, Execute:=(AutoFlow=10 OR AutoFlow=201) AND bInterlockXY, Position:=OilPointY, Velocity:=HMI_AutoSpeedXY, Acceleration:=HMI_Acc,Deceleration:=HMI_Dec,jerk:=HMI_Jerk);		//Go Oil
MC_MoveAbsolute3(Axis:=MC_AxisZ, Execute:=AutoFlow=20 AND bInterlockZ, Position:=OilPointZ, Velocity:=HMI_AutoSpeedZ);		//Go Oil
MC_MoveAbsolute4(Axis:=MC_AxisX, Execute:=(AutoFlow=400) AND bInterlockXY, Position:=0, Velocity:=HMI_AutoSpeedXY, Acceleration:=HMI_Acc,Deceleration:=HMI_Dec,jerk:=HMI_Jerk);		//Go 0
MC_MoveAbsolute5(Axis:=MC_AxisY, Execute:=(AutoFlow=400) AND bInterlockXY, Position:=0, Velocity:=HMI_AutoSpeedXY, Acceleration:=HMI_Acc,Deceleration:=HMI_Dec,jerk:=HMI_Jerk);		//Go 0
MC_MoveAbsolute6(Axis:=MC_AxisZ, Execute:=(AutoFlow=40 OR AutoFlow=300) AND bInterlockZ, Position:=0, Velocity:=HMI_AutoSpeedZ);		//Go 0
MC_MoveAbsolute7(Axis:=MC_AxisX, Execute:=AutoFlow=100 AND bInterlockXY, Position:=ScrewDatas[HMI_JobNo].PositionX[HMI_PointNo], Velocity:=HMI_AutoSpeedXY, Acceleration:=HMI_Acc,Deceleration:=HMI_Dec,jerk:=HMI_Jerk);		//Go ABS
MC_MoveAbsolute8(Axis:=MC_AxisY, Execute:=AutoFlow=100 AND bInterlockXY, Position:=ScrewDatas[HMI_JobNo].PositionY[HMI_PointNo], Velocity:=HMI_AutoSpeedXY, Acceleration:=HMI_Acc,Deceleration:=HMI_Dec,jerk:=HMI_Jerk);		//Go ABS
MC_MoveAbsolute9(Axis:=MC_AxisZ, Execute:=AutoFlow=103 AND bInterlockZ, Position:=ScrewDatas[HMI_JobNo].PositionZ[HMI_PointNo], Velocity:=HMI_AutoSpeedZ);		//Go ABS

ErrorState:=
Error_AxisX OR
Error_AxisY OR
Error_AxisZ  OR
Error_PB_ESTOP;
//********************************************************************
//power on =0
IF NOT(SystemReadyStatus) OR ErrorState OR NOT(AutoStatus) THEN
	AutoFlow:=0;
	MachineRunning:=FALSE;
	Main2FeedScrewFlag:=FALSE;
	Main2DownFlag:=FALSE;
	Main2UpFlag:=FALSE;
	Main2ScrewFlag:=FALSE;
	ResetFeedScrewErrorFlag:=FALSE;
END_IF;
//idle=1
IF AutoFlow=0 AND SystemReadyStatus AND NOT(ErrorState) AND AutoStatus THEN
	AutoFlow:=1;
END_IF;
IF AutoFlow=203 AND NOT(PB_Start) AND HMI_PointNo=0 THEN
	MachineRunning:=FALSE;
	HMI_AllCount:=HMI_AllCount+1;
	AutoFlow:=1;
END_IF;
IF AutoFlow=405 AND NOT(SOL_Fix) AND Error_SNR_FeedScrew THEN
	MachineRunning:=FALSE;
	AutoFlow:=1;
END_IF;
//start,clear HMI show data=2
R_TRIG1(Clk:=PB_Start);
IF R_TRIG1.Q THEN
	RunStatus:=TRUE;
END_IF;
IF ErrorState OR AutoFlow=0 OR Error_LS_UpDownBack OR Error_LS_UpDownOut OR PB_Reset THEN
	RunStatus:=FALSE;
END_IF;
IF AutoFlow=1 AND R_TRIG1.Q AND NOT(Error_SNR_AirSource) AND NOT(Error_SNR_FeedScrew) AND NOT(Error_LS_THBack) AND NOT(Error_LS_THOut) THEN
	FOR iv:=0 TO 29 BY 1 DO
	    ShowOKs[iv]:=FALSE;
		ShowNGs[iv]:=FALSE;
	END_FOR;
	//HMI_PointNo:=0;
	feedcount:=0;
	MachineRunning:=TRUE;
	AutoFlow:=2;
END_IF;
//x,y go to oil point=10
IF AutoFlow=2 AND SOL_Fix THEN
	AutoFlow:=10;
END_IF;
//moving=11
IF AutoFlow=10 AND (MC_MoveAbsolute1.Active OR MC_MoveAbsolute2.Active) THEN
	AutoFlow:=11;
END_IF;
//reached=12
IF AutoFlow=11 AND NOT(MC_MoveAbsolute1.Active) AND NOT(MC_MoveAbsolute2.Active) THEN
	AutoFlow:=12;
END_IF;
//z go to oil point=20
IF AutoFlow=12 THEN
	AutoFlow:=20;
END_IF;
//moving=21
IF AutoFlow=20 AND MC_MoveAbsolute3.Active THEN
	AutoFlow:=21;
END_IF;
//reached=22
IF AutoFlow=21 AND NOT(MC_MoveAbsolute3.Active) THEN
	AutoFlow:=22;
END_IF;
//sol down=30
IF AutoFlow=22 AND MC_AxisZ.Status.Standstill THEN
	Main2DownFlag:=TRUE;
	AutoFlow:=30;
END_IF;
//sol up=31
TON1(In:=(AutoFlow=30 OR AutoFlow=403) AND LS_UpDownOut , PT:=t#500ms);
IF AutoFlow=30 AND TON1.Q THEN
	Main2DownFlag:=FALSE;
	Main2UpFlag:=TRUE;
	AutoFlow:=31;
END_IF;
//z go to 0=40
IF AutoFlow=31 AND LS_UpDownBack THEN
	Main2UpFlag:=FALSE;
	AutoFlow:=40;
END_IF;
IF AutoFlow=108 THEN
	AutoFlow:=40;
END_IF;
//moving=41
IF AutoFlow=40 AND MC_MoveAbsolute6.Active THEN
	AutoFlow:=41;
END_IF;
//reached=42
IF AutoFlow=41 AND NOT(MC_MoveAbsolute6.Active) THEN
	AutoFlow:=42;
END_IF;
//check is last point?=43
IF AutoFlow=42 THEN
	AutoFlow:=43;
END_IF;
IF AutoFlow=404 AND LS_UpDownBack AND feedcount<3 THEN
	AutoFlow:=43;
	Main2UpFlag:=FALSE;
END_IF;
//********************************************************************
//not last point.=50
IF AutoFlow=43 AND NOT(ScrewDatas[HMI_JobNo].IsLastPoint[HMI_PointNo]) THEN
	AutoFlow:=50;
END_IF;
//Feed screw start=51
IF AutoFlow=50 AND RunStatus AND NOT(Main2FeedScrewFlag) THEN
	IF HMI_PointNo<>0 THEN
		Main2FeedScrewFlag:=TRUE;
	END_IF;
	AutoFlow:=51;
END_IF;
//Feed screw done=52
IF AutoFlow=51 AND (Main2FeedScrewFlag OR HMI_PointNo=0) THEN
	AutoFlow:=52;
END_IF;
//x,y go to screw point=100
IF AutoFlow=52 THEN
	AutoFlow:=100;
END_IF;
//moving=101
IF AutoFlow=100 AND (MC_MoveAbsolute7.Active OR MC_MoveAbsolute8.Active) THEN
	AutoFlow:=101;
END_IF;
//reached=102
IF AutoFlow=101 AND NOT(MC_MoveAbsolute7.Active) AND NOT(MC_MoveAbsolute8.Active) THEN
	
	AutoFlow:=102;
END_IF;
//z go to screw point=103
IF AutoFlow=102 THEN
	IF HMI_PointNo=0 THEN
		Main2FeedScrewFlag:=TRUE;
	END_IF;
	AutoFlow:=103;
END_IF;
//moving=104
IF AutoFlow=103 AND MC_MoveAbsolute9.Active AND (Main2FeedScrewFlag OR HMI_PointNo<>0) THEN
	AutoFlow:=104;
END_IF;
//reached=105
IF AutoFlow=104 AND NOT(MC_MoveAbsolute9.Active) THEN
	AutoFlow:=105;
END_IF;
//********************************************************************
//call screw start=106
TON3(In:=AutoFlow=105 AND NOT(Main2FeedScrewFlag), PT:=t#100ms);
IF AutoFlow=105 AND NOT(FeedScrewErrorFlag) AND TON3.Q THEN
	Main2ScrewFlag:=TRUE;
	AutoFlow:=106;
END_IF;
//screw done=107
//TON2(In:=Main2FeedScrewFlag, PT:=NanoSecToTime(HMI_FeedScrewTime*100000000));
//IF TON2.Q THEN
	//Main2FeedScrewFlag:=FALSE;
//END_IF;
IF AutoFlow=106 AND NOT(Main2ScrewFlag) THEN
	feedcount:=0;
	AutoFlow:=107;
END_IF;
//point no. add 1=108
IF AutoFlow=107 AND feedcount=0 THEN
	HMI_PointNo:=HMI_PointNo+1;
	AutoFlow:=108;
END_IF;
//********************************************************************
//is last point.=200
IF AutoFlow=43 AND (ScrewDatas[HMI_JobNo].IsLastPoint[HMI_PointNo]) THEN
	AutoFlow:=200;
END_IF;
//x,y go to 0=201
IF AutoFlow=200 THEN
	AutoFlow:=201;
END_IF;
//moving=202
IF AutoFlow=201 AND (MC_MoveAbsolute1.Active OR MC_MoveAbsolute2.Active) THEN
	AutoFlow:=202;
END_IF;
//reached,point no. set 0=203
IF AutoFlow=202 AND NOT(SOL_Fix) AND NOT(MC_MoveAbsolute1.Active) AND NOT(MC_MoveAbsolute2.Active) THEN
	HMI_PointNo:=0;
	FOR jValue:=0 TO 29 BY 1 DO
	    IF ShowNGs[jValue] THEN
		    ScrewNGFlag:=TRUE;
		END_IF;
	END_FOR;
	AutoFlow:=203;
END_IF;
TON4(In:=ScrewNGFlag,PT:=t#1s);
IF TON4.Q THEN
	ScrewNGFlag:=FALSE;
END_IF;
//********************************************************************
IF PB_Reset THEN
	Error_SNR_FeedScrew:=FALSE;
END_IF;
//z go to 0=300
IF AutoFlow=105 AND (FeedScrewErrorFlag) AND TON3.Q THEN
	AutoFlow:=300;
	feedcount:=feedcount+1;
	ResetFeedScrewErrorFlag:=TRUE;
END_IF;
//moving=301
IF AutoFlow=300 AND MC_MoveAbsolute6.Active THEN
	AutoFlow:=301;
END_IF;
//reached=302
IF AutoFlow=301 AND NOT(FeedScrewErrorFlag) AND NOT(MC_MoveAbsolute6.Active) THEN
	AutoFlow:=302;
	ResetFeedScrewErrorFlag:=FALSE;
END_IF;
//x,y go to 0=400
IF AutoFlow=302 AND NOT(ResetFeedScrewErrorFlag) THEN
	AutoFlow:=400;
END_IF;
//moving=401
IF AutoFlow=400 AND (MC_MoveAbsolute4.Active OR MC_MoveAbsolute5.Active) THEN
	AutoFlow:=401;
END_IF;
//reached=402
IF AutoFlow=401 AND NOT(MC_MoveAbsolute4.Active) AND NOT(MC_MoveAbsolute5.Active) THEN
	AutoFlow:=402;
END_IF;
//sol down=403
IF AutoFlow=402 THEN
	Main2DownFlag:=TRUE;
	AutoFlow:=403;
END_IF;
//sol up=404
IF AutoFlow=403 AND TON1.Q THEN
	AutoFlow:=404;
	Main2DownFlag:=FALSE;
	Main2UpFlag:=TRUE;
END_IF;
//set error=405
IF AutoFlow=404 AND LS_UpDownBack AND feedcount>=3 THEN
	AutoFlow:=405;
	Main2UpFlag:=FALSE;
	Error_SNR_FeedScrew:=TRUE;
END_IF;
END_PROGRAM

PROGRAM prScrewFlow
VAR
    fbSol1 : SingleSolRy;
    fbSol2 : SingleSolRy;
    AutoFlow : INT;
    ErrorState : BOOL;
    TON1 : TON;
    TON2 : TON;
    TON3 : TON;
    MC_TorqueControl1 : MC_TorqueControl;
    TorqueValue : LREAL;
    SpeedValue : LREAL;
    tCheckNGTime : TIME;
    tCheckOKTime : TIME;
    MC_MoveRelative1 : MC_MoveRelative;
END_VAR
VAR_EXTERNAL
    HMIPB_UpDown : BOOL;
    AutoStatus : BOOL;
    SOL_UpDown : BOOL;
    SystemReadyStatus : BOOL;
END_VAR
VAR_EXTERNAL CONSTANT
    MC_AxisZ : _sAXIS_REF;
    MC_AxisX : _sAXIS_REF;
    MC_AxisY : _sAXIS_REF;
END_VAR
VAR_EXTERNAL
    LS_UpDownBack : BOOL;
    UP_InitialFlag : BOOL;
    Error_LS_UpDownBack : BOOL;
    Error_LS_UpDownOut : BOOL;
    Main2ScrewFlag : BOOL;
    SNR_InPositionCheck : BOOL;
    ScrewStopFlag : BOOL;
    HMIPB_ScrewMode_Torque : BOOL;
    HMIPB_AlarmResetAxisS : BOOL;
END_VAR
VAR_EXTERNAL CONSTANT
    MC_AxisS : _sAXIS_REF;
END_VAR
VAR_EXTERNAL
    HMI_ScrewTorque : LREAL;
    HMI_ScrewSpeed : LREAL;
    ScrewDatas : array[0..39] of stscrewdata;
    ShowOKs : ARRAY[0..29] of bool;
    HMI_PointNo : INT;
    ShowNGs : ARRAY[0..29] of bool;
    Error_PB_ESTOP : BOOL;
    Error_AxisS : BOOL;
    HMI_CheckNGTime : LINT;
    HMI_CheckOKTime : LINT;
    Main2DownFlag : BOOL;
    Main2UpFlag : BOOL;
    Main2FeedScrewFlag : BOOL;
    HMI_BackoutD : LREAL;
END_VAR
//********************************************************************
//Manual
//********************************************************************
//up and down sol
fbSol1(
	HMIPB_UpDown,
	AutoStatus,
	AutoFlow=2 OR Main2DownFlag,
	AutoFlow=4 OR UP_InitialFlag OR Main2UpFlag,
	TRUE,
	MC_AxisX.Details.Homed AND MC_AxisX.Status.Standstill AND MC_AxisY.Details.Homed AND MC_AxisY.Status.Standstill,
	SOL_UpDown);
//********************************************************************
//Auto
//power on=0
//idle=1
//start,sol down=2
//axis s start=3
//Axis s screwing=500

//reach sensor,axis s stop=100
// not reach sensor time's up,axis s stop=200

//torque ok,axis s stop=300
//torque ng,axis s stop=400

//sol up=4
//sol reach up,finish=5
//********************************************************************
ErrorState:=
Error_AxisS OR
Error_PB_ESTOP;
//power on=0
IF NOT(SystemReadyStatus) OR ErrorState THEN
	AutoFlow:=0;
END_IF;
//idle=1
IF AutoFlow=0 AND SystemReadyStatus AND NOT(ErrorState) THEN
	AutoFlow:=1;
END_IF;
IF AutoFlow=5 AND NOT(Main2ScrewFlag) THEN
	AutoFlow:=1;
END_IF;
//start,sol down=2
IF AutoFlow=1 AND Main2ScrewFlag THEN
	AutoFlow:=2;
END_IF;
//axis s start=3
IF AutoFlow=2 AND SOL_UpDown AND NOT(LS_UpDownBack) THEN
	AutoFlow:=3;
END_IF;
TorqueValue:=HMI_ScrewTorque;
SpeedValue:=HMI_ScrewSpeed/360;
MC_TorqueControl1(Axis:=MC_AxisS, Execute:=AutoFlow=3, Torque:=TorqueValue, TorqueRamp:=0, Velocity:=SpeedValue, Direction:=_mcPositiveDirection, BufferMode:=_mcAborting);
//Axis s screwing=500
IF AutoFlow=3 AND MC_TorqueControl1.Active THEN
	AutoFlow:=500;
END_IF;

//reach sensor,axis s stop=100
IF AutoFlow=500 AND NOT(HMIPB_ScrewMode_Torque) AND SNR_InPositionCheck THEN
	AutoFlow:=100;
	ShowOKs[HMI_PointNo]:=TRUE;
	ScrewStopFlag:=TRUE;
END_IF;

// not reach sensor time's up,axis s stop=200
tCheckNGTime:=NanoSecToTime(In:=HMI_CheckNGTime*100000000);
TON1(In:=AutoFlow=500 AND NOT(SNR_InPositionCheck), PT:=tCheckNGTime);
IF AutoFlow=500 AND NOT(HMIPB_ScrewMode_Torque) AND TON1.Q THEN
	AutoFlow:=200;
	ShowNGs[HMI_PointNo]:=TRUE;
	ScrewStopFlag:=TRUE;
END_IF;

//torque ok,axis s stop=300
tCheckOKTime:=NanoSecToTime(In:=HMI_CheckOKTime*100000000);
TON2(In:=AutoFlow=500 AND MC_TorqueControl1.InTorque, PT:=tCheckOKTime);
IF AutoFlow=500 AND (HMIPB_ScrewMode_Torque) AND TON2.Q THEN
	AutoFlow:=300;
	ShowOKs[HMI_PointNo]:=TRUE;
	ScrewStopFlag:=TRUE;
END_IF;

//torque ng,axis s stop=400
TON3(In:=AutoFlow=500 AND NOT(TON2.Q), PT:=tCheckNGTime);
IF AutoFlow=500 AND (HMIPB_ScrewMode_Torque) AND TON3.Q THEN
	AutoFlow:=400;
	ShowNGs[HMI_PointNo]:=TRUE;
	ScrewStopFlag:=TRUE;
END_IF;
//axis s stoping=600
IF (AutoFlow=100 OR AutoFlow=300) AND MC_AxisS.Status.Stopping THEN
	AutoFlow:=600;
	ScrewStopFlag:=FALSE;
END_IF;
//axis s stoped=601
IF AutoFlow=600 AND NOT(ScrewStopFlag) AND MC_AxisS.Status.Standstill THEN
	AutoFlow:=601;
END_IF;
//axis s backout=602
IF AutoFlow=601 THEN
	AutoFlow:=602;
END_IF;
MC_MoveRelative1(Axis:=MC_AxisS, Execute:=AutoFlow=602, Distance:=HMI_BackoutD, Velocity:=HMI_ScrewSpeed, BufferMode:=_mcAborting);
//axis s moving=603
IF AutoFlow=602 AND MC_MoveRelative1.Active THEN
	AutoFlow:=603;
END_IF;
//axis s moved=604
IF AutoFlow=603 AND NOT(MC_MoveRelative1.Active) THEN
	AutoFlow:=604;
END_IF;
//sol up=4
IF AutoFlow=604 AND MC_AxisS.Status.Standstill THEN
	AutoFlow:=4;
	ScrewStopFlag:=FALSE;
END_IF;
IF AutoFlow=200 AND MC_AxisS.Status.Stopping THEN
	AutoFlow:=4;
	ScrewStopFlag:=FALSE;
END_IF;
IF AutoFlow=400  AND MC_AxisS.Status.Stopping THEN
	AutoFlow:=4;
	ScrewStopFlag:=FALSE;
END_IF;
//sol reach up,finish=5
IF AutoFlow=4 AND LS_UpDownBack THEN
	AutoFlow:=5;
	Main2ScrewFlag:=FALSE;
END_IF;
END_PROGRAM

PROGRAM prFeedScrew
VAR
    fbSol3 : SingleSolRy;
    fbSol4 : SingleSolRy;
    ErrorState : BOOL;
    AutoFlow : INT;
    TON1 : TON;
    TON2 : TON;
    TON3 : TON;
    TON4 : TON;
    Check1 : fbCheckScrew_Clamp;
    TON5 : TON;
    testbit1 : BOOL;
END_VAR
VAR_EXTERNAL
    AutoStatus : BOOL;
    HMIPB_TH : BOOL;
    SOL_TH : BOOL;
    HMIPB_FeedScrew : BOOL;
    SOL_FeedScrew : BOOL;
    LS_THBack : BOOL;
    LS_THOut : BOOL;
    SystemReadyStatus : BOOL;
    Main2FeedScrewFlag : BOOL;
    HMI_FeedScrewTime : LINT;
    LS_UpDownOut : BOOL;
    SNR_FeedScrew : BOOL;
    ScrewInClip : INT;
    PB_Reset : BOOL;
    Error_SNR_FeedScrew : BOOL;
    Error_LS_THBack : BOOL;
    Error_LS_THOut : BOOL;
    FeedScrewErrorFlag : BOOL;
    ResetFeedScrewErrorFlag : BOOL;
END_VAR
//********************************************************************
//Check
//********************************************************************
Check1(
	inClearSingle:=LS_UpDownOut,
	inFeedSNR:=SNR_FeedScrew,
	inBlowSOL:=SOL_FeedScrew,
	inReset:=PB_Reset OR ResetFeedScrewErrorFlag,
	outError=>FeedScrewErrorFlag,
	inoutScrewInClip:=ScrewInClip);
//********************************************************************
//Manual
//********************************************************************
//TH sol
fbSol3(
	HMIPB_TH,
	AutoStatus,
	AutoFlow=4,
	AutoFlow=5,
	TRUE,
	TRUE,
	SOL_TH);
//Feed screw sol
fbSol4(
	HMIPB_FeedScrew,
	AutoStatus,
	AutoFlow=2,
	AutoFlow=3,
	TRUE,
	TRUE,
	SOL_FeedScrew);
//********************************************************************
//Auto
//power on=0
//idle=1
//feed screw on=2
//feed screw off=3
//th on=4
//th off=5
//********************************************************************
ErrorState:=
Error_LS_THBack OR
Error_LS_THOut;
//power on=0
IF NOT(SystemReadyStatus) OR ErrorState THEN
	AutoFlow:=0;
	Main2FeedScrewFlag:=FALSE;
END_IF;
//idle=1
IF AutoFlow=0 AND NOT(NOT(SystemReadyStatus) OR ErrorState) THEN
	AutoFlow:=1;
END_IF;
TON3(In:=AutoFlow=5, PT:=t#1s);
TON5(In:=AutoFlow=5 AND LS_THBack, PT:=t#500ms);
IF AutoFlow=5 AND (TON5.Q OR TON3.Q) THEN
	AutoFlow:=1;
	
END_IF;
//feed screw on=2
IF AutoFlow=1 AND Main2FeedScrewFlag THEN
	AutoFlow:=2;
END_IF;
//feed screw off=3
TON1(In:=AutoFlow=2 AND SOL_FeedScrew, PT:=NanoSecToTime(HMI_FeedScrewTime*100000000));
IF AutoFlow=2 AND TON1.Q THEN
	AutoFlow:=3;
END_IF;
//th on=4
IF AutoFlow=3 AND NOT(SOL_FeedScrew) THEN
	AutoFlow:=4;
	Main2FeedScrewFlag:=FALSE;
END_IF;
//th off=5
TON2(In:=AutoFlow=4 AND LS_THOut, PT:=t#1s);
TON4(In:=AutoFlow=4 AND NOT(LS_THOut), PT:=t#2s);
IF AutoFlow=4 AND (TON4.Q OR TON2.Q) THEN
	AutoFlow:=5;
END_IF;
END_PROGRAM

FUNCTION_BLOCK BowlFeeder
VAR
    AutoFlow : INT;
    TON_Auto1 : TON;
    TON_Auto2 : TON;
    TON_Auto3 : TON;
    tItemNotExistDelayTime : TIME;
    tItemExistTime : TIME;
    tItemNotExistErrorTime : TIME;
END_VAR
VAR_INPUT
    bFullSNR : BOOL;
    iItemNotExistDelayTime : LINT;
    iItemExistTime : LINT;
    iItemNotExistErrorTime : LINT;
END_VAR
VAR_OUTPUT
    bFullRY : BOOL;
    bFullSNRError : BOOL;
END_VAR
VAR_EXTERNAL
    SystemReadyStatus : BOOL;
END_VAR
(******************************************************************
程式:振動筒程序
作者:蔡相偉
版本資訊:v1.0		2016/4/16
******************************************************************)
//時間轉換
tItemNotExistDelayTime:=NanoSecToTime(In:=iItemNotExistDelayTime*100000000);
tItemExistTime:=NanoSecToTime(In:=iItemExistTime*100000000);
tItemNotExistErrorTime:=NanoSecToTime(In:=iItemNotExistErrorTime*100000000);
(*流程*)
(*PowerOn=0*)
IF NOT(SystemReadyStatus) THEN
	AutoFlow:=0;
END_IF;

(*Idle=1*)
IF AutoFlow=0 AND SystemReadyStatus THEN
	AutoFlow:=1;
END_IF;

IF AutoFlow=3 THEN
	AutoFlow:=1;
END_IF;

(*振動筒起振=2*)
TON_Auto1(IN:=AutoFlow=1 AND NOT(bFullSNR) , PT:=tItemNotExistDelayTime);
IF AutoFlow=1 AND TON_Auto1.Q THEN
	AutoFlow:=2;
END_IF;

(*振動筒停振=3*)
TON_Auto2(IN:=AutoFlow=2 AND bFullSNR , PT:=tItemExistTime);
TON_Auto3(IN:=NOT(bFullSNR) AND bFullRY, PT:=tItemNotExistErrorTime);
IF AutoFlow=2 AND TON_Auto2.Q THEN
	AutoFlow:=3;
END_IF;
(******************************************************************)
(*輸出*)
(*振動筒繼電器*)
IF AutoFlow=2 THEN
	bFullRY:=TRUE;
	ELSE
	bFullRY:=FALSE;
END_IF;
(*振動筒滿料異常*)
IF AutoFlow=2 AND (TON_Auto3.Q) THEN
	bFullSNRError:=TRUE;
	ELSE
	bFullSNRError:=FALSE;
END_IF;
END_FUNCTION_BLOCK

FUNCTION_BLOCK SingleSolRy
VAR
    solStatus : BOOL;
    R_TRIG1 : R_TRIG;
END_VAR
VAR_INPUT
    inPushButton : BOOL;
    inAutoStatus : BOOL;
    inAutoFlowSet : BOOL;
    inAutoFlowReset : BOOL;
    inInterLockBack : BOOL;
    inInterLockOut : BOOL;
END_VAR
VAR_OUTPUT
    outSol : BOOL;
END_VAR
(*電磁閥*)
R_TRIG1(Clk:=inPushButton AND NOT(inAutoStatus));
(*SET*)
IF ((R_TRIG1.Q AND NOT(solStatus)) OR inAutoFlowSet) AND inInterLockOut THEN
	outSol:=TRUE;
END_IF;
(*RESET*)
IF ((R_TRIG1.Q AND (solStatus)) OR inAutoFlowReset) AND inInterLockBack THEN
	outSol:=FALSE;
END_IF;
(*STATUS*)
solStatus:=outSol;
END_FUNCTION_BLOCK

FUNCTION_BLOCK fbErrorSOL_S
VAR
    TON_1 : TON;
    TON_2 : TON;
END_VAR
VAR_INPUT
    bAutoStatus : BOOL;
    bResetPB : BOOL;
    bSOL : BOOL;
    bBackLS : BOOL;
    bOutLS : BOOL;
END_VAR
VAR_OUTPUT
    bErrorStatus_Back : BOOL;
    bErrorStatus_Out : BOOL;
END_VAR
IF bAutoStatus AND NOT(bResetPB) THEN
	(*歸磁簧開關*)
	TON_1(IN:=(NOT(bSOL) AND NOT(bBackLS)) OR ((bSOL) AND bBackLS), PT:=t#2s);
	IF TON_1.Q THEN
		bErrorStatus_Back:=TRUE;
	END_IF;
	(*出磁簧開關*)
	TON_2(IN:=(NOT(bSOL) AND (bOutLS)) OR ((bSOL) AND NOT(bOutLS)), PT:=t#2s);
	IF TON_2.Q THEN
		bErrorStatus_Out:=TRUE;
	END_IF;
END_IF;
IF bResetPB THEN
	bErrorStatus_Back:=FALSE;
	bErrorStatus_Out:=FALSE;
END_IF;
END_FUNCTION_BLOCK

FUNCTION_BLOCK fbErrorSOL_D
VAR
    TON_1 : TON;
    TON_2 : TON;
END_VAR
VAR_INPUT
    bAutoStatus : BOOL;
    bResetPB : BOOL;
    bBackSOL : BOOL;
    bOutSOL : BOOL;
    bBackLS : BOOL;
    bOutLS : BOOL;
END_VAR
VAR_OUTPUT
    bErrorStatus_Back : BOOL;
    bErrorStatus_Out : BOOL;
END_VAR
IF bAutoStatus AND NOT(bResetPB) THEN
	(*歸磁簧開關*)
	TON_1(IN:=bBackSOL AND NOT(bBackLS), PT:=t#4s);
	IF TON_1.Q THEN
		bErrorStatus_Back:=TRUE;
	END_IF;
	(*出磁簧開關*)
	TON_2(IN:=bOutSOL AND NOT(bOutLS), PT:=t#4s);
	IF TON_2.Q THEN
		bErrorStatus_Out:=TRUE;
	END_IF;
END_IF;
IF bResetPB THEN
	bErrorStatus_Back:=FALSE;
	bErrorStatus_Out:=FALSE;
END_IF;
END_FUNCTION_BLOCK

FUNCTION_BLOCK fbCheckScrew_Clamp
VAR
    R_TRIG1 : R_TRIG;
    R_TRIG2 : R_TRIG;
    F_TRIG1 : F_TRIG;
END_VAR
VAR_INPUT
    inClearSingle : BOOL;
    inFeedSNR : BOOL;
    inBlowSOL : BOOL;
    inReset : BOOL;
END_VAR
VAR_OUTPUT
    outError : BOOL;
END_VAR
VAR_IN_OUT
    inoutScrewInClip : INT;
END_VAR
R_TRIG1(CLK:= inClearSingle);
R_TRIG2(CLK:= inFeedSNR);
F_TRIG1(Clk:=inBlowSOL);

IF R_TRIG2.Q THEN
	inoutScrewInClip:=inoutScrewInClip+1;
END_IF;

IF R_TRIG1.Q THEN
	inoutScrewInClip:=0;
END_IF;

IF F_TRIG1.Q AND inoutScrewInClip<=0 THEN
	outError:=TRUE;
END_IF;
IF inReset THEN
	outError:=FALSE;
END_IF;
END_FUNCTION_BLOCK